(*********************************** G.D S.p.A. - Technical Department ***********************************
============= PROGRAM INFO ============
FOLDER:             TBD
MACHINES INVOLVED:  TBD 

============= DESCRIPTION =============
csp machine declaration

============= REVISIONS ===============
Date		Version	 	Author      	Description             
----------	-------		------------  	--------------------------------------------
2019/04/05 	0000.00	 	M.Grasso		Creation of the PRG

**********************************************************************************************************)
(*$R process_ref := prc; $*)
PROGRAM csp_case_glue_hotMelt_safety
VAR
	
	prc:											process;
	prc_path:										STRING;
	
	sig:											safety_integrated_group;
	sis:											safety_integrated_series;
END_VAR

_read_var_input();

_object_manager();

IF NOT objects_running()
THEN
	RETURN;	
END_IF

_read_process_image();

_mode_manager();

CASE process_get_mode(prc) of
	MODE_ABSENT,
	MODE_INACTIVE:
		RETURN;
	MODE_TEST:
		_handle_process_test();
END_CASE

_set_runtime_properties();

(********************************* BODY *********************************)
safety_integrated_series_close(sis);
(************************************************************************)

_handle_messages();

_write_output();

ACTION _handle_messages:
;
END_ACTION

ACTION _handle_process_test:
;
END_ACTION

ACTION _mode_manager:
IF process_mode_req_is_pending(prc)
THEN
    process_apply_mode_req_first_step(prc);
    CASE process_get_mode(prc) OF
        MODE_TO_ABSENT:
			;
        MODE_TO_INACTIVE:
			;
        MODE_TO_TEST:
			;
        MODE_TO_OPERATIONAL:
			;
    END_CASE
    process_apply_mode_req_second_step(prc);
END_IF
END_ACTION

ACTION _object_manager:
IF objects_initialization()
THEN
	sub_process_init(
		object_name						:= 'csp_case_glue_ls_guns_safety.prc', 
		process							:= csp_case_glue_ls_guns.prc, 
		CONVERSION_this					:= prc);
		
	prc_path 							:= process_get_path(prc);
	

END_IF

IF objects_running()
THEN
	process_cycle(prc);
	
END_IF
END_ACTION

ACTION _read_process_image:
;
END_ACTION

ACTION _read_var_input:
;
END_ACTION

ACTION _set_runtime_properties:
;
END_ACTION

ACTION _write_output:
;
END_ACTION

END_PROGRAM

(* stored: Version 1.1.0.1, ProductVersion 3.1.4024.3
   POU csp_case_glue_hotMelt_safety: Id {4a6d7ecf-e102-49cf-8b5e-70be00500f2f}, SpecialFunc None
   Action _handle_messages: Id {2a87ebd4-2f49-4f9a-a5d1-03ffb132bfab}
   Action _handle_process_test: Id {13d53cdf-80c2-407c-8fb5-d1f8ef58dded}
   Action _mode_manager: Id {de839279-390d-40f3-ba80-67e01793e28f}
   Action _object_manager: Id {a2030559-9618-46d3-b325-185a625b98f5}
   Action _read_process_image: Id {83bc1c25-3560-4272-b0d5-a374b8ca00f7}
   Action _read_var_input: Id {6cbf10b3-4458-46fd-a8b4-56ea8be23db1}
   Action _set_runtime_properties: Id {1d24a4e3-5672-403e-8213-9bdc7e008f80}
   Action _write_output: Id {fbff8052-6509-472c-9993-d44d755f7307} *)
